(* LS Electric XG5000 project: PRACTICE *)
(* PLC LSPLC *)

PROGRAM Q1. (* task: 스캔 프로그램 *)
VAR
    P1 : BOOL;
    P10 : BOOL;
    P11 : BOOL;
END_VAR

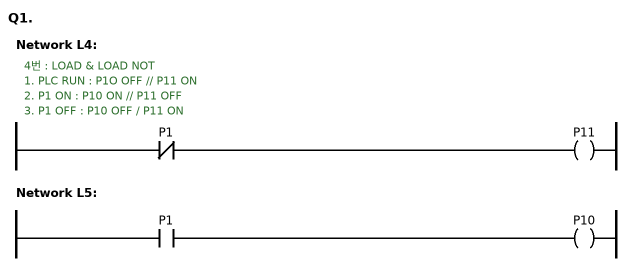
(* 4번 : LOAD & LOAD NOT *)
(* 1. PLC RUN : P1O OFF // P11 ON *)
(* 2. P1 ON : P10 ON // P11 OFF *)
(* 3. P1 OFF : P10 OFF / P11 ON *)
(* Rung L4 *)
P11 := NOT P1;
(* Rung L5 *)
P10 := P1;
END_PROGRAM

PROGRAM Q2 (* task: 스캔 프로그램 *)
VAR
    P1 : BOOL;
    P10 : BOOL;
END_VAR
VAR
    _e1 : R_TRIG;
END_VAR

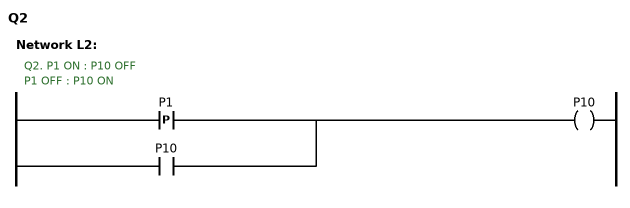
(* Q2. P1 ON : P10 OFF *)
(* P1 OFF : P10 ON *)
(* Rung L2 *)
_e1(CLK := P1);
P10 := _e1.Q OR P10;
END_PROGRAM

PROGRAM Q3. (* task: 스캔 프로그램 *)
VAR
    P1 : BOOL;
    P10 : BOOL;
    P2 : BOOL;
END_VAR
VAR
    _e1 : R_TRIG;
    _e2 : R_TRIG;
END_VAR

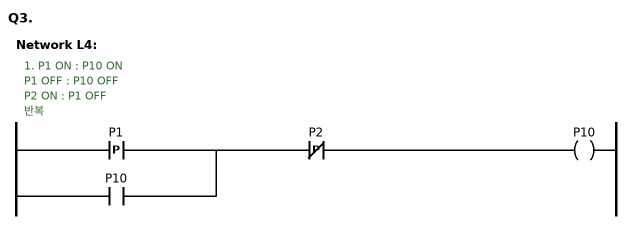
(* 1. P1 ON : P10 ON *)
(* P1 OFF : P10 OFF *)
(* P2 ON : P1 OFF *)
(* 반복 *)
(* Rung L4 *)
_e1(CLK := P1);
_e2(CLK := P2);
P10 := (_e1.Q OR P10) AND NOT _e2.Q;
END_PROGRAM

PROGRAM Q4. (* task: 스캔 프로그램 *)
VAR
    P1 : BOOL;
    P10 : BOOL;
    P2 : BOOL;
    P3 : BOOL;
END_VAR
VAR
    _e1 : R_TRIG;
    _e2 : R_TRIG;
END_VAR

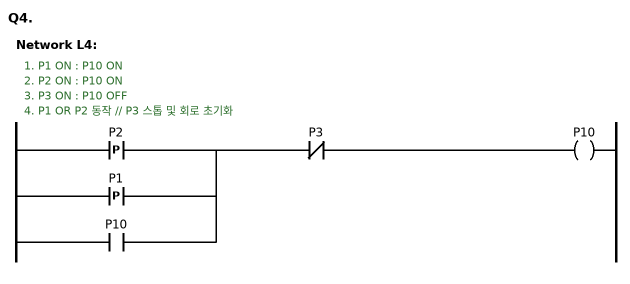
(* 1. P1 ON : P10 ON *)
(* 2. P2 ON : P10 ON *)
(* 3. P3 ON : P10 OFF *)
(* 4. P1 OR P2 동작 // P3 스톱 및 회로 초기화 *)
(* Rung L4 *)
_e1(CLK := P2);
_e2(CLK := P1);
P10 := (_e1.Q OR _e2.Q OR P10) AND NOT P3;
END_PROGRAM

PROGRAM Q5. (* task: 스캔 프로그램 *)
VAR
    P1 : BOOL;
    P10 : BOOL;
    P11 : BOOL;
    P2 : BOOL;
    P3 : BOOL;
END_VAR
VAR
    _e1 : R_TRIG;
    _e2 : R_TRIG;
    _e3 : R_TRIG;
END_VAR

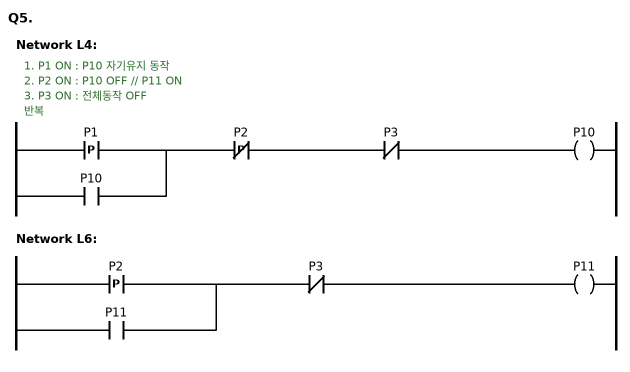
(* 1. P1 ON : P10 자기유지 동작 *)
(* 2. P2 ON : P10 OFF // P11 ON *)
(* 3. P3 ON : 전체동작 OFF *)
(* 반복 *)
(* Rung L4 *)
_e1(CLK := P1);
_e2(CLK := P2);
P10 := (_e1.Q OR P10) AND NOT _e2.Q AND NOT P3;
(* Rung L6 *)
_e3(CLK := P2);
P11 := (_e3.Q OR P11) AND NOT P3;
END_PROGRAM

PROGRAM Q6. (* task: 스캔 프로그램 *)
VAR
    FLAG : BOOL;
    FLAG2 : BOOL;
    P1 : BOOL;
    P10 : BOOL;
    P11 : BOOL;
    P12 : BOOL;
    P2 : BOOL;
    P3 : BOOL;
END_VAR
VAR
    _e1 : R_TRIG;
    _e2 : R_TRIG;
    _e3 : R_TRIG;
    _e4 : R_TRIG;
END_VAR

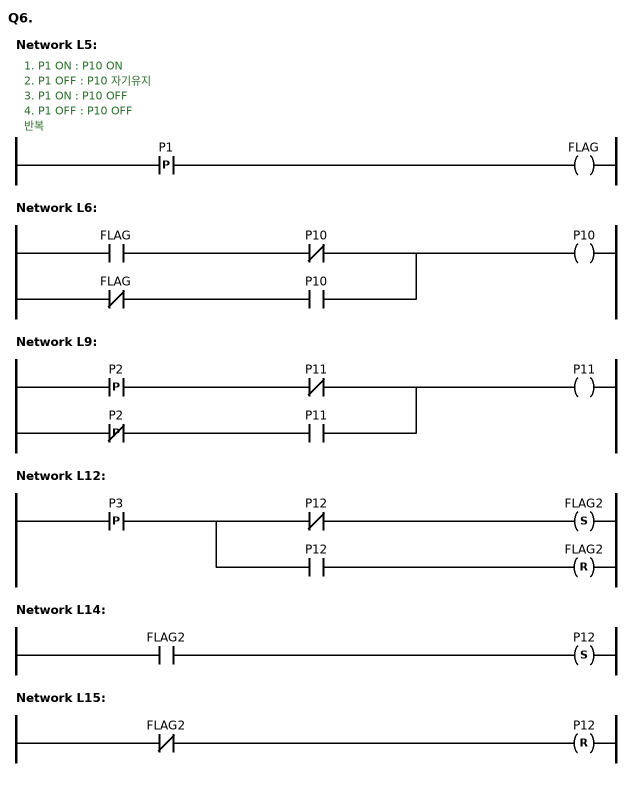
(* 1. P1 ON : P10 ON *)
(* 2. P1 OFF : P10 자기유지 *)
(* 3. P1 ON : P10 OFF *)
(* 4. P1 OFF : P10 OFF *)
(* 반복 *)
(* Rung L5 *)
_e1(CLK := P1);
FLAG := _e1.Q;
(* Rung L6 *)
P10 := (FLAG AND NOT P10) OR (NOT FLAG AND P10);
(* Rung L9 *)
_e2(CLK := P2);
_e3(CLK := P2);
P11 := (_e2.Q AND NOT P11) OR (NOT _e3.Q AND P11);
(* Rung L12 *)
_e4(CLK := P3);
IF _e4.Q AND NOT P12 THEN FLAG2 := TRUE; END_IF;
IF _e4.Q AND P12 THEN FLAG2 := FALSE; END_IF;
(* Rung L14 *)
IF FLAG2 THEN P12 := TRUE; END_IF;
(* Rung L15 *)
IF NOT FLAG2 THEN P12 := FALSE; END_IF;
END_PROGRAM

PROGRAM Q7. (* task: 스캔 프로그램 *)
VAR
    P0 : BOOL;
    P10 : BOOL;
    T0 : TON;
END_VAR

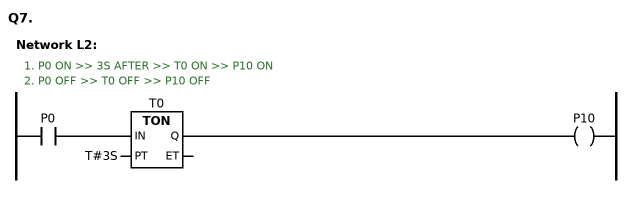
(* 1. P0 ON >> 3S AFTER >> T0 ON >> P10 ON *)
(* 2. P0 OFF >> T0 OFF >> P10 OFF *)
(* Rung L2 *)
T0(IN := P0, PT := T#3S);
P10 := T0.Q;
END_PROGRAM

PROGRAM Q8. (* task: 스캔 프로그램 *)
VAR
    P1 : BOOL;
    P10 : BOOL;
    P2 : BOOL;
    T0 : TON;
END_VAR

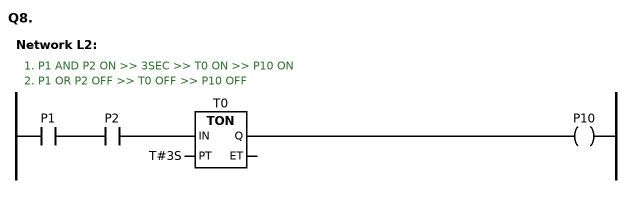
(* 1. P1 AND P2 ON >> 3SEC >> T0 ON >> P10 ON *)
(* 2. P1 OR P2 OFF >> T0 OFF >> P10 OFF *)
(* Rung L2 *)
T0(IN := P1 AND P2, PT := T#3S);
P10 := T0.Q;
END_PROGRAM

PROGRAM Q9. (* task: 스캔 프로그램 *)
VAR
    FLAG : BOOL;
    P1 : BOOL;
    P10 : BOOL;
    STOP : BOOL;
    T1 : TON_UINT;
    T2 : TP;
END_VAR
VAR
    _e1 : R_TRIG;
END_VAR

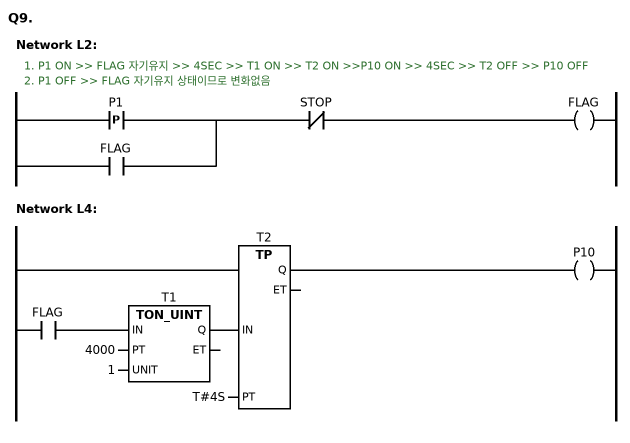
(* 1. P1 ON >> FLAG 자기유지 >> 4SEC >> T1 ON >> T2 ON >>P10 ON >> 4SEC >> T2 OFF >> P10 OFF *)
(* 2. P1 OFF >> FLAG 자기유지 상태이므로 변화없음 *)
(* Rung L2 *)
_e1(CLK := P1);
FLAG := (_e1.Q OR FLAG) AND NOT STOP;
(* Rung L4 *)
T1(IN := FLAG, PT := 4000, UNIT := 1);
T2(IN := T1.Q, PT := T#4S);
P10 := T2.Q;
END_PROGRAM

PROGRAM Q10. (* task: 스캔 프로그램 *)
VAR
    P1 : BOOL;
    P10 : BOOL;
    T1 : TP;
    T2 : TP;
END_VAR

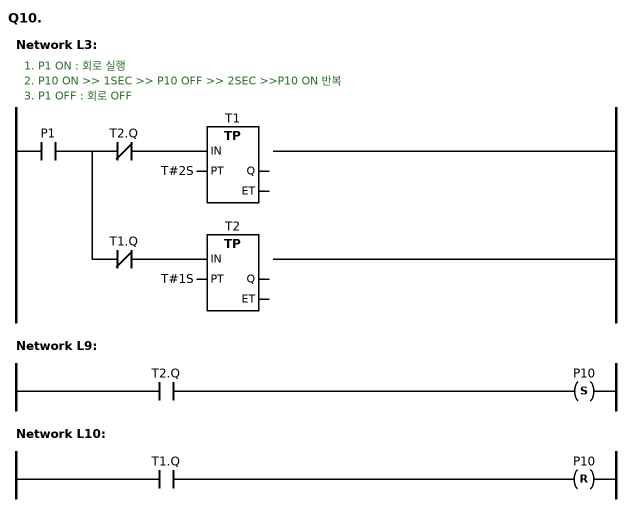
(* 1. P1 ON : 회로 실행 *)
(* 2. P10 ON >> 1SEC >> P10 OFF >> 2SEC >>P10 ON 반복 *)
(* 3. P1 OFF : 회로 OFF *)
(* Rung L3 *)
T1(IN := P1 AND NOT T2.Q, PT := T#2S);
T2(IN := P1 AND NOT T1.Q, PT := T#1S);
(* Rung L9 *)
IF T2.Q THEN P10 := TRUE; END_IF;
(* Rung L10 *)
IF T1.Q THEN P10 := FALSE; END_IF;
END_PROGRAM

PROGRAM Q11. (* task: 스캔 프로그램 *)
VAR
    P1 : BOOL;
    P10 : BOOL;
    P11 : BOOL;
    P12 : BOOL;
    T1 : TON;
    T2 : TON;
    T3 : TON;
END_VAR
VAR
    _e1 : R_TRIG;
END_VAR

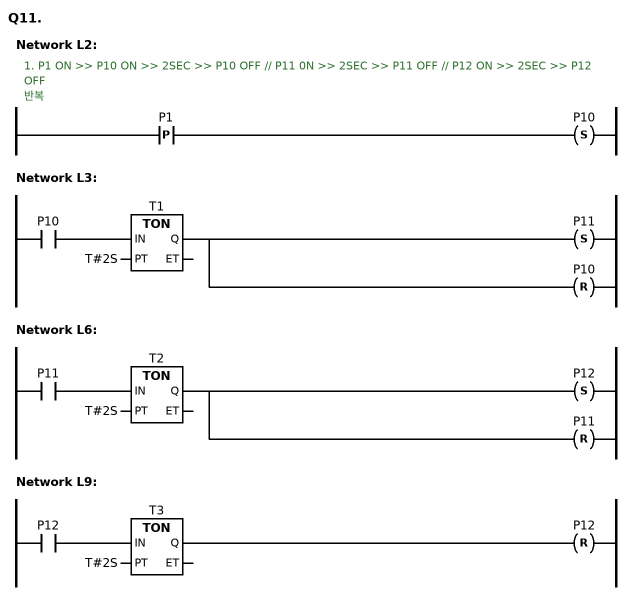
(* 1. P1 ON >> P10 ON >> 2SEC >> P10 OFF // P11 0N >> 2SEC >> P11 OFF // P12 ON >> 2SEC >> P12 OFF *)
(* 반복 *)
(* Rung L2 *)
_e1(CLK := P1);
IF _e1.Q THEN P10 := TRUE; END_IF;
(* Rung L3 *)
T1(IN := P10, PT := T#2S);
IF T1.Q THEN
    P11 := TRUE;
    P10 := FALSE;
END_IF;
(* Rung L6 *)
T2(IN := P11, PT := T#2S);
IF T2.Q THEN
    P12 := TRUE;
    P11 := FALSE;
END_IF;
(* Rung L9 *)
T3(IN := P12, PT := T#2S);
IF T3.Q THEN P12 := FALSE; END_IF;
END_PROGRAM

PROGRAM Q12. (* task: 스캔 프로그램 *)
VAR
    CV : INT;
    FUN : CTU_INT;
    P1 : BOOL;
    P10 : BOOL;
    P2 : BOOL;
    PV : INT := 4;
END_VAR
VAR
    _e1 : R_TRIG;
    _e2 : R_TRIG;
END_VAR

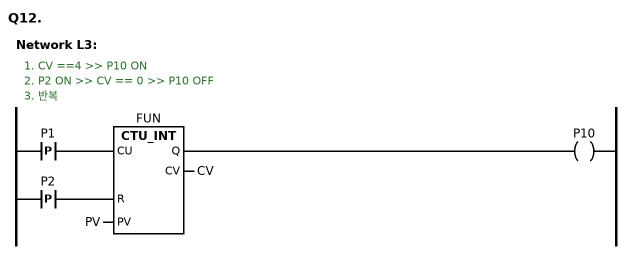
(* 1. CV ==4 >> P10 ON *)
(* 2. P2 ON >> CV == 0 >> P10 OFF *)
(* 3. 반복 *)
(* Rung L3 *)
_e1(CLK := P1);
_e2(CLK := P2);
FUN(CU := _e1.Q, R := _e2.Q, PV := PV, CV => CV);
P10 := FUN.Q;
END_PROGRAM

PROGRAM Q13. (* task: 스캔 프로그램 *)
VAR
    CV : INT;
    CV2 : INT;
    FUN : CTU_INT;
    INST : CTU_INT;
    P1 : BOOL;
    P10 : BOOL;
    P11 : BOOL;
    P12 : BOOL;
    P13 : BOOL;
    P2 : BOOL;
    PV : INT := 3;
    PV2 : INT := 3;
    R : BOOL;
    RESET : BOOL;
END_VAR
VAR
    _e1 : R_TRIG;
    _e2 : R_TRIG;
    _e3 : R_TRIG;
    _e4 : R_TRIG;
END_VAR

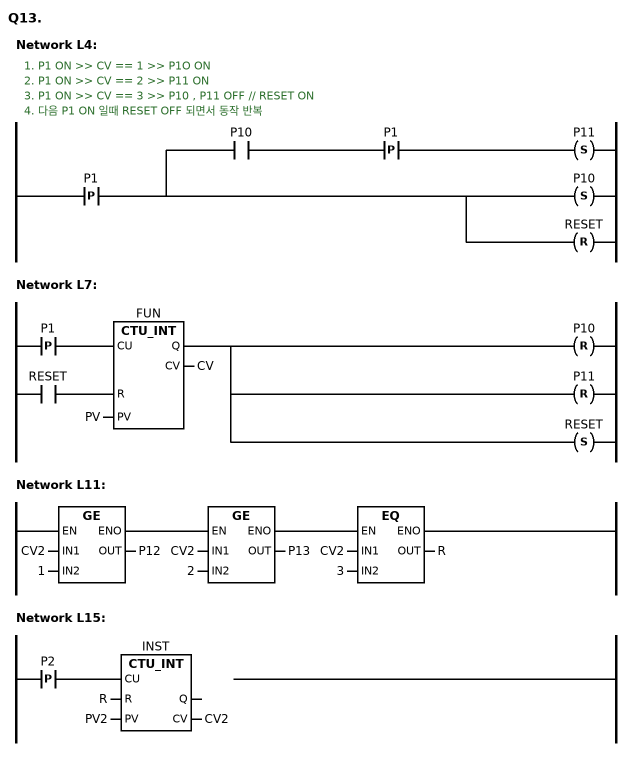
(* 1. P1 ON >> CV == 1 >> P1O ON *)
(* 2. P1 ON >> CV == 2 >> P11 ON *)
(* 3. P1 ON >> CV == 3 >> P10 , P11 OFF // RESET ON *)
(* 4. 다음 P1 ON 일때 RESET OFF 되면서 동작 반복 *)
(* Rung L4 *)
_e1(CLK := P1);
_e2(CLK := P1);
IF _e1.Q AND P10 AND _e2.Q THEN P11 := TRUE; END_IF;
IF _e1.Q THEN
    P10 := TRUE;
    RESET := FALSE;
END_IF;
(* Rung L7 *)
_e3(CLK := P1);
FUN(CU := _e3.Q, R := RESET, PV := PV, CV => CV);
IF FUN.Q THEN
    P10 := FALSE;
    P11 := FALSE;
    RESET := TRUE;
END_IF;
(* Rung L11 *)
P12 := CV2 >= 1;
P13 := CV2 >= 2;
R := CV2 = 3;
(* Rung L15 *)
_e4(CLK := P2);
INST(CU := _e4.Q, R := R, PV := PV2, CV => CV2);
END_PROGRAM